FUNCTION_BLOCK RunDevices
VAR_INPUT
END_VAR
VAR_OUTPUT
END_VAR
VAR
	device : POINTER TO ExecuteBase;
	command AT%I* : BYTE;
	acknowledge AT%Q* : BYTE;
	
	commandAsEnum : eCylinderCommands;
END_VAR

//------------
//	Bridger
//------------
//internalCommand := command;

CASE command OF
	0:
		commandAsEnum := eCylinderCommands.NO_COMMAND;
	1:
		commandAsEnum := eCylinderCommands.COMMAND_A;
	2:
		commandAsEnum := eCylinderCommands.COMMAND_B;
END_CASE
 
IF device<>0 AND_THEN device^.Execute(commandAsEnum) THEN
	acknowledge := command;
END_IF

METHOD FB_init : BOOL
VAR_INPUT
	bInitRetains : BOOL; // if TRUE, the retain variables are initialized (warm start / cold start)
	bInCopyCode : BOOL;  // if TRUE, the instance afterwards gets moved into the copy code (online change)

	argDevice : POINTER TO ExecuteBase;
END_VAR
device := argDevice;
END_METHOD

END_FUNCTION_BLOCK

(* stored: Version 1.1.0.1, ProductVersion 3.1.4024.0
   POU RunDevices: Id {8da684a8-fee9-4e71-99ee-14497b4e0900}, SpecialFunc None
   Method FB_init: Id {2559ac98-23b7-4255-9fdd-6cd997e5ed3d} *)
